(* PLC project Gen3Safety, BrAutomation SafeDESIGNER  5.19.0.0 *)
(* stored: companyURL http://www.br-automation.com, creationDateTime Fri Jun 14 14:03:41 2024 *)

PROGRAM Main
  VAR  (* added by the conversion: wires and edge detectors of the diagram *)
    _AND_S638_OUT : ANY;
    _SAFEBOOL_TO_BOOL637_OUT : BOOL;
    _BOOL_TO_SAFEBOOL457_OUT : SAFEBOOL;
    _BOOL_TO_SAFEBOOL460_OUT : SAFEBOOL;
    _BOOL_TO_SAFEBOOL466_OUT : SAFEBOOL;
    _BOOL_TO_SAFEBOOL469_OUT : SAFEBOOL;
  END_VAR

(* FBD diagram, written out as Structured Text *)
RackEnableBits(IN := VFLCRRacksEnabled);
Rack2Enabled := RackEnableBits.OUT_1;
Rack1Enabled := RackEnableBits.OUT_0;
Rack4Enabled := RackEnableBits.OUT_3;
Rack3Enabled := RackEnableBits.OUT_2;
_AND_S638_OUT := AND_S(SM41_OK, SM42_OK, SM43_OK, SM44_OK, Chiller1Running, Chiller2Running, EStopSafetyReset);
_SAFEBOOL_TO_BOOL637_OUT := SAFEBOOL_TO_BOOL(_AND_S638_OUT);
SM41_Release := _SAFEBOOL_TO_BOOL637_OUT;
enableReady := _AND_S638_OUT;
SM42_Release := _SAFEBOOL_TO_BOOL637_OUT;
SM44_Release := _SAFEBOOL_TO_BOOL637_OUT;
SM43_Release := _SAFEBOOL_TO_BOOL637_OUT;
status_SafetySystemReady := _AND_S638_OUT;
SF_EDM_ContactorLaserRack1(Activate := TRUE, S_OutControl := AND_S(enableReady, BOOL_TO_SAFEBOOL(cmd_EnableLaserSafety AND Rack1Enabled)), S_EDM1 := Rack1_PowerContactor_CH1_EDM, S_EDM2 := Rack1_PowerContactor_CH2_EDM, MonitoringTime := TIME#750ms, S_StartReset := SAFEFALSE, Reset := cmd_RequestLaserSafetyReset);
FBK_Error_EDMRack1 := SF_EDM_ContactorLaserRack1.Error;
FBK_Diag_EDMRack1 := SF_EDM_ContactorLaserRack1.DiagCode;
Rack1_PowerContactor_CH1 := SF_EDM_ContactorLaserRack1.S_EDM_Out;
Rack1_PowerContactor_CH2 := SF_EDM_ContactorLaserRack1.S_EDM_Out;
TON_S_DelayVFLCRSafety1(IN := AND_S(Rack1_PowerContactor_CH1, Rack1_PowerContactor_CH2), PT := SAFETIME#4s);
SF_EDM_SafetyRelayVFLCR1(Activate := TRUE, S_OutControl := TON_S_DelayVFLCRSafety1.Q, S_EDM1 := VFLCR1_SafetyRelay_EDM, S_EDM2 := VFLCR1_SafetyRelay_EDM, MonitoringTime := TIME#500ms, S_StartReset := SAFETRUE, Reset := cmd_RequestLaserSafetyReset);
VFLCR1_SafetyRelay_CH1 := SF_EDM_SafetyRelayVFLCR1.S_EDM_Out;
VFLCR1_SafetyRelay_CH2 := SF_EDM_SafetyRelayVFLCR1.S_EDM_Out;
SF_EDM_ContactorLaserRack2(Activate := TRUE, S_OutControl := AND_S(enableReady, BOOL_TO_SAFEBOOL(cmd_EnableLaserSafety AND Rack2Enabled)), S_EDM1 := Rack2_PowerContactor_CH1_EDM, S_EDM2 := Rack2_PowerContactor_CH2_EDM, MonitoringTime := TIME#750ms, S_StartReset := SAFEFALSE, Reset := cmd_RequestLaserSafetyReset);
FBK_Error_EDMRack2 := SF_EDM_ContactorLaserRack2.Error;
FBK_Diag_EDMRack2 := SF_EDM_ContactorLaserRack2.DiagCode;
Rack2_PowerContactor_CH1 := SF_EDM_ContactorLaserRack2.S_EDM_Out;
Rack2_PowerContactor_CH2 := SF_EDM_ContactorLaserRack2.S_EDM_Out;
TON_S_DelayVFLCRSafety2(IN := AND_S(Rack2_PowerContactor_CH1, Rack2_PowerContactor_CH2), PT := SAFETIME#4s);
SF_EDM_SafetyRelayVFLCR2(Activate := TRUE, S_OutControl := TON_S_DelayVFLCRSafety2.Q, S_EDM1 := VFLCR2_SafetyRelay_EDM, S_EDM2 := VFLCR2_SafetyRelay_EDM, MonitoringTime := TIME#500ms, S_StartReset := SAFETRUE, Reset := cmd_RequestLaserSafetyReset);
VFLCR2_SafetyRelay_CH1 := SF_EDM_SafetyRelayVFLCR2.S_EDM_Out;
VFLCR2_SafetyRelay_CH2 := SF_EDM_SafetyRelayVFLCR2.S_EDM_Out;
SF_EDM_ContactorLaserRack3(Activate := TRUE, S_OutControl := AND_S(enableReady, BOOL_TO_SAFEBOOL(cmd_EnableLaserSafety AND Rack3Enabled)), S_EDM1 := Rack3_PowerContactor_CH1_EDM, S_EDM2 := Rack3_PowerContactor_CH2_EDM, MonitoringTime := TIME#750ms, S_StartReset := SAFEFALSE, Reset := cmd_RequestLaserSafetyReset);
FBK_Error_EDMRack3 := SF_EDM_ContactorLaserRack3.Error;
FBK_Diag_EDMRack3 := SF_EDM_ContactorLaserRack3.DiagCode;
Rack3_PowerContactor_CH1 := SF_EDM_ContactorLaserRack3.S_EDM_Out;
Rack3_PowerContactor_CH2 := SF_EDM_ContactorLaserRack3.S_EDM_Out;
TON_S_DelayVFLCRSafety3(IN := AND_S(Rack3_PowerContactor_CH1, Rack3_PowerContactor_CH2), PT := SAFETIME#4s);
SF_EDM_SafetyRelayVFLCR3(Activate := TRUE, S_OutControl := TON_S_DelayVFLCRSafety3.Q, S_EDM1 := VFLCR3_SafetyRelay_EDM, S_EDM2 := VFLCR3_SafetyRelay_EDM, MonitoringTime := TIME#500ms, S_StartReset := SAFETRUE, Reset := cmd_RequestLaserSafetyReset);
VFLCR3_SafetyRelay_CH1 := SF_EDM_SafetyRelayVFLCR3.S_EDM_Out;
VFLCR3_SafetyRelay_CH2 := SF_EDM_SafetyRelayVFLCR3.S_EDM_Out;
SF_EDM_ContactorLaserRack4(Activate := TRUE, S_OutControl := AND_S(enableReady, BOOL_TO_SAFEBOOL(cmd_EnableLaserSafety AND Rack4Enabled)), S_EDM1 := Rack4_PowerContactor_CH1_EDM, S_EDM2 := Rack4_PowerContactor_CH2_EDM, MonitoringTime := TIME#750ms, S_StartReset := SAFEFALSE, Reset := cmd_RequestLaserSafetyReset);
FBK_Error_EDMRack4 := SF_EDM_ContactorLaserRack4.Error;
FBK_Diag_EDMRack4 := SF_EDM_ContactorLaserRack4.DiagCode;
Rack4_PowerContactor_CH1 := SF_EDM_ContactorLaserRack4.S_EDM_Out;
Rack4_PowerContactor_CH2 := SF_EDM_ContactorLaserRack4.S_EDM_Out;
TON_S_DelayVFLCRSafety4(IN := AND_S(Rack4_PowerContactor_CH1, Rack4_PowerContactor_CH2), PT := SAFETIME#4s);
SF_EDM_SafetyRelayVFLCR4(Activate := TRUE, S_OutControl := TON_S_DelayVFLCRSafety4.Q, S_EDM1 := VFLCR4_SafetyRelay_EDM, S_EDM2 := VFLCR4_SafetyRelay_EDM, MonitoringTime := TIME#500ms, S_StartReset := SAFETRUE, Reset := cmd_RequestLaserSafetyReset);
VFLCR4_SafetyRelay_CH1 := SF_EDM_SafetyRelayVFLCR4.S_EDM_Out;
VFLCR4_SafetyRelay_CH2 := SF_EDM_SafetyRelayVFLCR4.S_EDM_Out;
_BOOL_TO_SAFEBOOL457_OUT := BOOL_TO_SAFEBOOL(Rack1Enabled);
_BOOL_TO_SAFEBOOL460_OUT := BOOL_TO_SAFEBOOL(Rack2Enabled);
_BOOL_TO_SAFEBOOL466_OUT := BOOL_TO_SAFEBOOL(Rack3Enabled);
_BOOL_TO_SAFEBOOL469_OUT := BOOL_TO_SAFEBOOL(Rack4Enabled);
status_SafetyReset_Lasers := SAFEBOOL_TO_BOOL(AND_S(OR_S(AND_S(Rack1_PowerContactor_CH1, VFLCR1_SafetyRelay_CH1, _BOOL_TO_SAFEBOOL457_OUT), NOT_S(_BOOL_TO_SAFEBOOL457_OUT)), OR_S(AND_S(Rack2_PowerContactor_CH1, VFLCR2_SafetyRelay_CH1, _BOOL_TO_SAFEBOOL460_OUT), NOT_S(_BOOL_TO_SAFEBOOL460_OUT)), OR_S(AND_S(Rack3_PowerContactor_CH1, VFLCR3_SafetyRelay_CH1, _BOOL_TO_SAFEBOOL466_OUT), NOT_S(_BOOL_TO_SAFEBOOL466_OUT)), OR_S(AND_S(Rack4_PowerContactor_CH1, VFLCR4_SafetyRelay_CH1, _BOOL_TO_SAFEBOOL469_OUT), NOT_S(_BOOL_TO_SAFEBOOL469_OUT)))) AND NOT (NOT Rack1Enabled AND NOT Rack2Enabled AND NOT Rack3Enabled AND NOT Rack4Enabled);
status_FBK_Error_LaserEDM := FBK_Error_EDMRack1 OR FBK_Error_EDMRack2 OR FBK_Error_EDMRack3 OR FBK_Error_EDMRack4;
status_FBK_Diag_LaserEDM1 := FBK_Diag_EDMRack1;
status_FBK_Diag_LaserEDM2 := FBK_Diag_EDMRack2;
status_FBK_Diag_LaserEDM3 := FBK_Diag_EDMRack3;
status_FBK_Diag_LaserEDM4 := FBK_Diag_EDMRack4;
status_FBKERR_LaserEDM1 := FBK_Error_EDMRack1;
status_FBKERR_LaserEDM2 := FBK_Error_EDMRack2;
status_FBKERR_LaserEDM3 := FBK_Error_EDMRack3;
status_FBKERR_LaserEDM4 := FBK_Error_EDMRack4;
END_PROGRAM
